(* IEC 61131-3 sources: xPLCCore/codesys_code/Application/COMM_FBs/FB_MpUnpacker, 14 files *)

(* ---- TryReadINTBuffer.st ---- *)
FUNCTION TryReadINTBuffer : POINTER TO BYTE
VAR_INPUT
	sPath 	: STRING; 				  // Path to the integer value
	p_data_size : POINTER TO INT;     // Pointer to an INT to store the size (1, 2, 4, or 8 bytes)
	p_signedness : POINTER TO BOOL;   // Pointer to a BOOL to store if it's signed (TRUE) or unsigned (FALSE)
END_VAR
VAR
	pValue 	: POINTER TO BYTE;    // Pointer to the start of the MessagePack value (type byte)
	tmpByte : BYTE;               // To hold the MessagePack type byte
END_VAR
(* =========== IMPLEMENTATION =========== *)

	// Initialize outputs to default/error states
	IF p_data_size <> 0 THEN
		p_data_size^ := 0; // Default size to 0
	END_IF;
	IF p_signedness <> 0 THEN
		p_signedness^ := FALSE; // Default signedness to FALSE (unsigned)
	END_IF;
	TryReadINTBuffer := 0; // Default return to NULL pointer (no integer found/decoded)

	// Attempt to find the value by path
	IF NOT FindValueByPath(sPath, pValue) THEN
		RETURN; // Value not found, return NULL pointer and default output parameters
	END_IF;

	// Check for NULL pointer from FindValueByPath (should be handled by NOT condition above, but good defense)
	IF pValue = 0 THEN
		RETURN;
	END_IF;

	tmpByte := pValue^; // Read the MessagePack type byte

	// Determine integer type, size, and signedness based on the type byte
	CASE tmpByte OF
		// --- Positive Fixint (0x00 - 0x7F) ---
		0..16#7F: // 0xxxxxxx
			IF p_data_size <> 0 THEN p_data_size^ := 1; END_IF;
			IF p_signedness <> 0 THEN p_signedness^ := TRUE; END_IF; // Can be treated as signed
			TryReadINTBuffer := pValue; // Data is the type byte itself

		// --- Negative Fixint (0xE0 - 0xFF) ---
		16#E0..16#FF: // 111xxxxx
			IF p_data_size <> 0 THEN p_data_size^ := 1; END_IF;
			IF p_signedness <> 0 THEN p_signedness^ := TRUE; END_IF;
			TryReadINTBuffer := pValue; // Data is the type byte itself

		// --- Unsigned Integers ---
		16#CC: // uint 8
			IF p_data_size <> 0 THEN p_data_size^ := 1; END_IF;
			IF p_signedness <> 0 THEN p_signedness^ := FALSE; END_IF;
			TryReadINTBuffer := pValue + 1; // Data starts after the type byte

		16#CD: // uint 16
			IF p_data_size <> 0 THEN p_data_size^ := 2; END_IF;
			IF p_signedness <> 0 THEN p_signedness^ := FALSE; END_IF;
			TryReadINTBuffer := pValue + 1;

		16#CE: // uint 32
			IF p_data_size <> 0 THEN p_data_size^ := 4; END_IF;
			IF p_signedness <> 0 THEN p_signedness^ := FALSE; END_IF;
			TryReadINTBuffer := pValue + 1;

		16#CF: // uint 64
			IF p_data_size <> 0 THEN p_data_size^ := 8; END_IF;
			IF p_signedness <> 0 THEN p_signedness^ := FALSE; END_IF;
			TryReadINTBuffer := pValue + 1;

		// --- Signed Integers ---
		16#D0: // int 8
			IF p_data_size <> 0 THEN p_data_size^ := 1; END_IF;
			IF p_signedness <> 0 THEN p_signedness^ := TRUE; END_IF;
			TryReadINTBuffer := pValue + 1;

		16#D1: // int 16
			IF p_data_size <> 0 THEN p_data_size^ := 2; END_IF;
			IF p_signedness <> 0 THEN p_signedness^ := TRUE; END_IF;
			TryReadINTBuffer := pValue + 1;

		16#D2: // int 32
			IF p_data_size <> 0 THEN p_data_size^ := 4; END_IF;
			IF p_signedness <> 0 THEN p_signedness^ := TRUE; END_IF;
			TryReadINTBuffer := pValue + 1;

		16#D3: // int 64
			IF p_data_size <> 0 THEN p_data_size^ := 8; END_IF;
			IF p_signedness <> 0 THEN p_signedness^ := TRUE; END_IF;
			TryReadINTBuffer := pValue + 1;

		ELSE
			// If not an integer type, return NULL pointer and default output parameters
			// (already set at the beginning of the function)
			TryReadINTBuffer := 0;
	END_CASE;

(* ---- FB_MpUnpacker.st ---- *)
(*
================================================================================
 FB_MpUnpacker: MessagePack Unpacker/Parser with Path Query
================================================================================
This function block parses a MessagePack byte stream.

Instructions:
1. Create a Function Block named 'FB_MpUnpacker'.
2. Copy the main variable declarations into its declaration part.
3. Add each METHOD to the FB, copying the respective variable declarations
   and implementation code.

New Feature: Path Querying
- You can now directly read a value using a path string.
- Use dot notation for nested objects: 'obj.key'
- Use brackets for array indices: 'arr[0]'
- Example: 'data.measurements[2].value'

Key Feature:
- Alignment-Safe: Uses MEMUtils.MemCpy for reading DINT and REAL values
  to prevent memory access violation errors on sensitive hardware.
*)
FUNCTION_BLOCK FB_MpUnpacker
VAR_INPUT
END_VAR
VAR_OUTPUT
	eLastType 		: E_MpType;
	diLastDINT 		: DINT;
	rLastREAL 		: REAL;
	sLastString 	: STRING;
	uiLastCount 	: UINT;
END_VAR
VAR CONSTANT
	MAX_NESTING_DEPTH : INT := 16;
END_VAR
VAR
	pStart 			: POINTER TO BYTE;
	pCurrent 		: POINTER TO BYTE;
	udiSize 		: UDINT;
END_VAR
(* =========== IMPLEMENTATION =========== *)

(* ---- FindValueByPath.st ---- *)
METHOD PRIVATE FindValueByPath : BOOL
VAR_INPUT
	sPath		: STRING;
END_VAR
VAR_IN_OUT
	pResult		: POINTER TO BYTE;
END_VAR
VAR
	sRemainingPath : STRING(255) := sPath;
	sSegment : STRING(80);
	nSepPos, nBracketPos, nEndBracketPos, i, nTargetIndex, nCounter : DINT;
	nMapCount, nArrayCount : UINT;
	sKeyFound : STRING;
	fbTempUnpacker : FB_MpUnpacker;
	// Local pointer for cleaner dereferencing
	pWordLen : POINTER TO WORD; // Declared here
END_VAR
(* =========== IMPLEMENTATION =========== *)
	FindValueByPath := FALSE;
	pResult := pStart;

	WHILE LEN(sRemainingPath) > 0 DO
		IF LEFT(sRemainingPath, 1) <> '[' THEN // This path segment is a key (for a map)
			nSepPos := FIND(sRemainingPath, '.');
			nBracketPos := FIND(sRemainingPath, '[');

			IF nSepPos > 0 AND (nBracketPos = 0 OR nSepPos < nBracketPos) THEN
				sSegment := LEFT(sRemainingPath, DINT_TO_INT(nSepPos - 1));
			ELSIF nBracketPos > 0 AND (nSepPos = 0 OR nBracketPos < nSepPos) THEN
				sSegment := LEFT(sRemainingPath, DINT_TO_INT(nBracketPos - 1));
			ELSE
				sSegment := sRemainingPath;
			END_IF;

			// Handle map header based on marker
			IF (pResult^ >= 16#80 AND pResult^ <= 16#8F) THEN // fixmap
				nMapCount := pResult^ - 16#80;
				pResult := pResult + 1;
			ELSIF pResult^ = 16#DE THEN // map 16
				// --- BUG FIX FOR MAP HEADER ---
				// This was the part still causing issues.
				pWordLen := pResult + 1; // Point to the 2-byte length field
				Swap16To(pWordLen,ADR(nMapCount));
				pResult := pResult + 3; // Advance pointer by 1 (marker) + 2 (count bytes)
			ELSE
				// Current element is not a map, so path segment is invalid
				RETURN;
			END_IF;

			nCounter := 0; // Use nCounter to track if key is found, -1 if found
			FOR i := 1 TO nMapCount DO
				// Initialize a temporary unpacker for the key
				fbTempUnpacker.Init(pResult, udiSize - (pResult - pStart));
				fbTempUnpacker.UnpackNext(); // Unpack the key
				sKeyFound := fbTempUnpacker.sLastString; // Get the key string

				IF NOT SkipValue(pResult) THEN RETURN; END_IF; // pResult now points to the value

				IF sKeyFound = sSegment THEN
					nCounter := -1; // Key found, mark as -1 and exit loop
					EXIT;
				ELSE
					IF NOT SkipValue(pResult) THEN RETURN; END_IF; // Skip the value if key not found
				END_IF;
			END_FOR;

			IF nCounter <> -1 THEN RETURN; END_IF; // If key not found after loop, return FALSE

			sRemainingPath := RIGHT(sRemainingPath, DINT_TO_INT(LEN(sRemainingPath) - LEN(sSegment)));
		ELSE
			nEndBracketPos := FIND(sRemainingPath, ']');
			IF nEndBracketPos = 0 THEN RETURN; END_IF;

			// Extract the index string, e.g., "55" from "[55]"
			sSegment := MID(sRemainingPath, 2, DINT_TO_INT(nEndBracketPos - 2));
			nTargetIndex := STRING_TO_DINT(sSegment);

			// Handle array header based on marker
			IF (pResult^ >= 16#90 AND pResult^ <= 16#9F) THEN // fixarray
				nArrayCount := pResult^ - 16#90;
				pResult := pResult + 1;
			ELSIF pResult^ = 16#DC THEN // array 16
				// --- PREVIOUS BUG FIX FOR ARRAY ---
				pWordLen := pResult + 1; // Point to the 2-byte length field

				Swap16To(pWordLen,ADR(nArrayCount));
				pResult := pResult + 3; // Advance pointer by 1 (marker) + 2 (count bytes)
			ELSE
				// Current element is not an array, so path segment is invalid
				RETURN;
			END_IF;

			// Check if the target index is within the array bounds
			IF nTargetIndex >= DINT_TO_UINT(nArrayCount) THEN RETURN; END_IF;

			// Skip elements until the target index is reached
			FOR i := 0 TO nTargetIndex - 1 DO
				IF NOT SkipValue(pResult) THEN RETURN; END_IF;
			END_FOR;

			sRemainingPath := RIGHT(sRemainingPath, DINT_TO_INT(LEN(sRemainingPath) - nEndBracketPos));

		END_IF;

		IF LEN(sRemainingPath) > 0 AND LEFT(sRemainingPath, 1) = '.' THEN
			sRemainingPath := RIGHT(sRemainingPath, DINT_TO_INT(LEN(sRemainingPath) - 1));
		END_IF;
	END_WHILE;

	FindValueByPath := TRUE;

(* ---- GetValueSize.st ---- *)
METHOD PRIVATE GetValueSize : UDINT
VAR_INPUT
	pObjectStart : POINTER TO BYTE;
END_VAR
VAR
	pTemp : POINTER TO BYTE;
END_VAR
(* =========== IMPLEMENTATION =========== *)
	pTemp := pObjectStart;
	IF SkipValue(pTemp) THEN
		GetValueSize := pTemp - pObjectStart;
	ELSE
		GetValueSize := 0;
	END_IF;

(* ---- Init.st ---- *)
(* Method: Init - (Implementation is unchanged) *)
METHOD Init : BOOL
VAR_INPUT
	pData 		: POINTER TO BYTE;
	udiDataSize : UDINT;
END_VAR
(* =========== IMPLEMENTATION =========== *)
	IF pData = 0 OR udiDataSize = 0 THEN Init := FALSE; RETURN; END_IF;
	pStart 		:= pData;
	pCurrent 	:= pData;
	udiSize 	:= udiDataSize;
	Init 		:= TRUE;

(* ---- SkipValue.st ---- *)
(*
Method: SkipValue [FINAL CORRECTED ITERATIVE VERSION]
Description: Advances a given pointer past the next complete value in the stream.
             This robust iterative version uses a simple counter to avoid recursion
             and correctly handle all MessagePack types.
Return Type: BOOL (TRUE if successful)
*)
METHOD PRIVATE SkipValue : BOOL
VAR_IN_OUT
	pPos : POINTER TO BYTE;
END_VAR
VAR
	diItemsToSkip : DINT := 1; // Start by wanting to skip 1 top-level item.
	byMarker : BYTE;
	udiLength : UDINT;
	uiCount : UINT;
	pWordLen : POINTER TO WORD;

    pDwordLen 	: POINTER TO DWORD;
    udiCount32 	: UDINT;
END_VAR
(* =========== IMPLEMENTATION =========== *)
	WHILE diItemsToSkip > 0 DO
		// Boundary check for each item to be skipped
		IF pPos >= (pStart + udiSize) THEN
			SkipValue := FALSE;
			RETURN;
		END_IF;

		diItemsToSkip := diItemsToSkip - 1; // Consume one item from the "to-skip" list

		byMarker := pPos^; // Read the marker of the current item
		pPos := pPos + 1;  // Advance pointer past the marker

		CASE byMarker OF
    // Nil, Bool, FixInt (0-byte payload, pointer already advanced)
    16#C0, 16#C2, 16#C3: CONTINUE;

    // --- Fixed-size Payloads ---
    16#CC, 16#D0: pPos := pPos + 1; // uint 8, int 8
    16#CD, 16#D1: pPos := pPos + 2; // uint 16, int 16
    16#CE, 16#D2, 16#CA: pPos := pPos + 4; // uint 32, int 32, float 32
    16#CF, 16#D3, 16#CB: pPos := pPos + 8; // uint 64, int 64, float 64

    // --- String Types ---
    16#D9: // str 8
        udiLength := pPos^;
        pPos := pPos + 1 + udiLength;
    16#DA: // str 16
        pWordLen := pPos;
        Swap16To(pWordLen, ADR(udiLength)); // Assumes udiLength gets lower 16 bits
        pPos := pPos + 2 + udiLength;
    16#DB: // str 32
        pDwordLen := pPos;
        Swap32To(pDwordLen, ADR(udiLength)); // Assumes Swap32To helper exists
        pPos := pPos + 4 + udiLength;

    // --- Binary Types ---
    16#C4: // bin 8
        udiLength := pPos^;
        pPos := pPos + 1 + udiLength;
    16#C5: // bin 16
        pWordLen := pPos;
        Swap16To(pWordLen, ADR(udiLength));
        pPos := pPos + 2 + udiLength;
    16#C6: // bin 32
        pDwordLen := pPos;
        Swap32To(pDwordLen, ADR(udiLength));
        pPos := pPos + 4 + udiLength;

    // --- Extension Types ---
    16#D4: pPos := pPos + 2;  // fixext 1 (1-byte type + 1-byte data)
    16#D5: pPos := pPos + 3;  // fixext 2
    16#D6: pPos := pPos + 5;  // fixext 4
    16#D7: pPos := pPos + 9;  // fixext 8
    16#D8: pPos := pPos + 17; // fixext 16
    16#C7: // ext 8
        udiLength := pPos^;
        pPos := pPos + 1 + 1 + udiLength; // len(1) + type(1) + data
    16#C8: // ext 16
        pWordLen := pPos;
        Swap16To(pWordLen, ADR(udiLength));
        pPos := pPos + 2 + 1 + udiLength; // len(2) + type(1) + data
    16#C9: // ext 32
        pDwordLen := pPos;
        Swap32To(pDwordLen, ADR(udiLength));
        pPos := pPos + 4 + 1 + udiLength; // len(4) + type(1) + data

ELSE
    IF (byMarker <= 16#7F) THEN // positive fixint
        CONTINUE;
    ELSIF (byMarker >= 16#E0) THEN // negative fixint
        CONTINUE;

    // fixstr
    ELSIF (byMarker >= 16#A0 AND byMarker <= 16#BF) THEN
        udiLength := byMarker - 16#A0;
        pPos := pPos + udiLength;

    // --- Container Types (add children to skip list) ---
    ELSIF (byMarker >= 16#90 AND byMarker <= 16#9F) THEN // fixarray
        uiCount := byMarker - 16#90;
        diItemsToSkip := diItemsToSkip + uiCount;
    ELSIF (byMarker = 16#DC) THEN // array 16
        pWordLen := pPos;
        Swap16To(pWordLen, ADR(uiCount));
        pPos := pPos + 2;
        diItemsToSkip := diItemsToSkip + uiCount;
    ELSIF (byMarker = 16#DD) THEN // array 32
        pDwordLen := pPos;
        Swap32To(pDwordLen, ADR(udiCount32));
        pPos := pPos + 4;
        diItemsToSkip := diItemsToSkip + udiCount32;

    ELSIF (byMarker >= 16#80 AND byMarker <= 16#8F) THEN // fixmap
        uiCount := (byMarker - 16#80);
        diItemsToSkip := diItemsToSkip + (uiCount * 2);
    ELSIF (byMarker = 16#DE) THEN // map 16
        pWordLen := pPos;
        Swap16To(pWordLen, ADR(uiCount));
        pPos := pPos + 2;
        diItemsToSkip := diItemsToSkip + (uiCount * 2);
    ELSIF (byMarker = 16#DF) THEN // map 32
        pDwordLen := pPos;
        Swap32To(pDwordLen, ADR(udiCount32));
        pPos := pPos + 4;
        diItemsToSkip := diItemsToSkip + (udiCount32 * 2);
    ELSE
        // Unknown marker, cannot safely skip.
        SkipValue := FALSE;
        RETURN;
    END_IF;
END_CASE;

	END_WHILE;

	SkipValue := TRUE;

(* ---- TryReadBool.st ---- *)
METHOD TryReadBool : BOOL
VAR_INPUT
	sPath 	: STRING;
	default : BOOL;
END_VAR
VAR
	pValue : POINTER TO BYTE;
END_VAR
(* =========== IMPLEMENTATION =========== *)
	TryReadBool := default;

	IF FindValueByPath(sPath, pValue) THEN
		IF pValue^ = 16#C2 THEN
			TryReadBool := FALSE;
		ELSIF pValue^ = 16#C3 THEN
			TryReadBool := TRUE;
		END_IF;
	END_IF;

(* ---- TryReadINT64.st ---- *)
METHOD TryReadINT64 : LINT
VAR_INPUT
	sPath 	: STRING; 				// Path to the value
	default 	: LINT; 		// Default value if not found or cannot decode
END_VAR
VAR
	pValue 	: POINTER TO BYTE;
	pCurrent : POINTER TO BYTE; // Pointer to advance through the data
	tmpByte 	: BYTE;
	tmpSint 	: SINT; // For int 8
	tmpWord 	: WORD; // For uint 16, int 16
	tmpInt 	: INT;  // For int 16
	tmpDint 	: DINT; // For uint 32, int 32
	tmpUdint 	: UDINT; // For uint 32
	tmpLint 	: LINT; // For int 64
	tmpULint 	: ULINT; // For uint 64
	// tmpReal : REAL; // Not needed as floats are excluded
	// tmpLReal : LREAL; // Not needed as floats are excluded

	// Define MAX_LINT if not globally available
	cMAX_LINT : LINT := 9223372036854775807; // 2^63 - 1
END_VAR
(* =========== IMPLEMENTATION =========== *)

	TryReadINT64 := default; // Initialize with default value

	IF FindValueByPath(sPath, pValue) THEN
		pCurrent := pValue; // Start at the beginning of the value's data

		// Get the MessagePack type byte
		tmpByte := pCurrent^;
		pCurrent := pCurrent + 1; // Advance pointer past the type byte

		CASE tmpByte OF
			// --- Positive Fixint (0x00 - 0x7F) ---
			0..16#7F: // 0xxxxxxx: Positive Fixint (1 byte)
				TryReadINT64 := BYTE_TO_LINT(tmpByte);

			// --- Negative Fixint (0xE0 - 0xFF) ---
			16#E0..16#FF: // 111xxxxx: Negative Fixint (-32 to -1) (1 byte)
				tmpSint := BYTE_TO_SINT(tmpByte);
				TryReadINT64 := SINT_TO_LINT(tmpSint);

			// --- Unsigned Integers ---
			16#CC: // uint 8 (1 byte value)
				tmpByte := pCurrent^;
				TryReadINT64 := BYTE_TO_LINT(tmpByte);

			16#CD: // uint 16 (2 byte value)
				Swap16To(srcData:=pCurrent, dstData:=ADR(tmpWord));
				TryReadINT64 := WORD_TO_LINT(tmpWord);

			16#CE: // uint 32 (4 byte value)
				Swap32To(srcData:=pCurrent, dstData:=ADR(tmpUdint));
				TryReadINT64 := UDINT_TO_LINT(tmpUdint);

			16#CF: // uint 64 (8 byte value)
				Swap64To(srcData:=pCurrent, dstData:=ADR(tmpULint));
				// Rule: "except (UINT64 && top bit is 1)"
				// This means if tmpULint > MAX_LINT, it cannot be represented as LINT.
				IF tmpULint > cMAX_LINT THEN
					TryReadINT64 := default; // Value too large for signed 64-bit integer
				ELSE
					TryReadINT64 := ULINT_TO_LINT(tmpULint);
				END_IF;

			// --- Signed Integers ---
			16#D0: // int 8 (1 byte value)
				tmpSint := pCurrent^;
				TryReadINT64 := SINT_TO_LINT(tmpSint);

			16#D1: // int 16 (2 byte value)
				Swap16To(srcData:=pCurrent, dstData:=ADR(tmpInt));
				TryReadINT64 := INT_TO_LINT(tmpInt);

			16#D2: // int 32 (4 byte value)
				Swap32To(srcData:=pCurrent, dstData:=ADR(tmpDint));
				TryReadINT64 := DINT_TO_LINT(tmpDint);

			16#D3: // int 64 (8 byte value)
				Swap64To(srcData:=pCurrent, dstData:=ADR(tmpLint));
				TryReadINT64 := tmpLint; // It's already LINT

			// --- Floating-Point Numbers ---
			16#CA, // float 32
			16#CB: // float 64
				// Rule: "they will not read floating point number"
				TryReadINT64 := default; // Explicitly return default for floats

			ELSE
				// Handle other unsupported MessagePack types (string, array, map, nil, ext type)
				TryReadINT64 := default;
		END_CASE;
	END_IF;

(* ---- TryReadObject.st ---- *)
(*
Method: TryReadObject [NEW FEATURE]
Description: Finds a map or array at a given path and initializes a destination
             unpacker instance to represent that sub-object.
Return Type: BOOL (TRUE on success)
*)
METHOD TryReadObject : BOOL
VAR_INPUT
	sPath 	: STRING; 					// Path to the map or array
	pDest 	: POINTER TO FB_MpUnpacker;	// Pointer to the destination unpacker instance
END_VAR
VAR
	pValue : POINTER TO BYTE;
	udiObjectSize : UDINT;
END_VAR
(* =========== IMPLEMENTATION =========== *)
	TryReadObject := FALSE;
	IF pDest = 0 THEN RETURN; END_IF;

	IF FindValueByPath(sPath, pValue) THEN
		IF (pValue^ >= 16#80 AND pValue^ <= 16#8F) OR (pValue^ = 16#DE) OR
		   (pValue^ >= 16#90 AND pValue^ <= 16#9F) OR (pValue^ = 16#DC) THEN
			udiObjectSize := GetValueSize(pObjectStart := pValue);

			IF udiObjectSize > 0 THEN
				TryReadObject := pDest^.Init(pData := pValue, udiDataSize := udiObjectSize);
				TryReadObject:=TRUE;
			END_IF;
		END_IF;
	END_IF;

(* ---- TryReadREAL.st ---- *)
METHOD TryReadREAL : REAL
VAR_INPUT
	sPath 	: STRING; 				// Path to the value
	default 	: REAL; 		// Default value if not found or cannot decode
END_VAR
VAR
	pValue 	: POINTER TO BYTE;
	pCurrent : POINTER TO BYTE; // Pointer to advance through the data
	tmpByte 	: BYTE;
	tmpSint 	: SINT; // For int 8
	tmpWord 	: WORD; // For uint 16, int 16
	tmpInt 	: INT;  // For int 16
	tmpDint 	: DINT; // For uint 32, int 32
	tmpUdint 	: UDINT; // For uint 32
	tmpLint 	: LINT; // For uint 64, int 64
	tmpULint 	: ULINT; // For uint 64
	tmpReal 	: REAL; // For float 32
	tmpLReal 	: LREAL; // For float 64 (double precision)
END_VAR
(* =========== IMPLEMENTATION =========== *)

	TryReadREAL := default; // Initialize with default value

	IF FindValueByPath(sPath, pValue) THEN
		pCurrent := pValue; // Start at the beginning of the value's data

		// Get the MessagePack type byte
		tmpByte := pCurrent^;
		pCurrent := pCurrent + 1; // Advance pointer past the type byte

		// Use a CASE statement for clarity and extensiveness
		CASE tmpByte OF
			// --- Positive Fixint (0x00 - 0x7F) ---
			0..16#7F: // 0xxxxxxx: Positive Fixint (1 byte)
				// The value is directly in tmpByte (pCurrent-1, as pCurrent already advanced)
				TryReadREAL := BYTE_TO_REAL(tmpByte);

			// --- Negative Fixint (0xE0 - 0xFF) ---
			16#E0..16#FF: // 111xxxxx: Negative Fixint (-32 to -1) (1 byte)
				// Treat the byte as SINT (signed 8-bit integer) to get the negative value.
				// tmpByte already holds the value
				tmpSint := BYTE_TO_SINT(tmpByte); // This correctly casts the byte's bits as a signed SINT
				TryReadREAL := SINT_TO_REAL(tmpSint);

			// --- Unsigned Integers ---
			16#CC: // uint 8 (1 byte value)
				tmpByte := pCurrent^; // Read the 1-byte unsigned integer
				TryReadREAL := BYTE_TO_REAL(tmpByte);
				// pCurrent will be implicitly advanced by the next loop iteration or return.

			16#CD: // uint 16 (2 byte value)
				Swap16To(srcData:=pCurrent, dstData:=ADR(tmpWord)); // Swap into tmpWord
				TryReadREAL := WORD_TO_REAL(tmpWord);
				// pCurrent := pCurrent + SIZEOF(WORD); // Already handled implicitly by FindValueByPath or next call

			16#CE: // uint 32 (4 byte value)
				Swap32To(srcData:=pCurrent, dstData:=ADR(tmpUdint)); // Swap into tmpUdint
				TryReadREAL := UDINT_TO_REAL(tmpUdint);
				// pCurrent := pCurrent + SIZEOF(UDINT); // Already handled implicitly

			16#CF: // uint 64 (8 byte value)
				Swap64To(srcData:=pCurrent, dstData:=ADR(tmpULint)); // Swap into tmpULint
				// Conversion from ULINT to REAL might lose precision for very large numbers
				TryReadREAL := ULINT_TO_REAL(tmpULint);
				// pCurrent := pCurrent + SIZEOF(ULINT); // Already handled implicitly

			// --- Signed Integers ---
			16#D0: // int 8 (1 byte value)
				tmpSint := pCurrent^; // Read the 1-byte signed integer
				TryReadREAL := SINT_TO_REAL(tmpSint);
				// pCurrent := pCurrent + SIZEOF(SINT); // Already handled implicitly

			16#D1: // int 16 (2 byte value)
				Swap16To(srcData:=pCurrent, dstData:=ADR(tmpInt)); // Swap into tmpInt
				TryReadREAL := INT_TO_REAL(tmpInt);
				// pCurrent := pCurrent + SIZEOF(INT); // Already handled implicitly

			16#D2: // int 32 (4 byte value)
				Swap32To(srcData:=pCurrent, dstData:=ADR(tmpDint)); // Swap into tmpDint
				TryReadREAL := DINT_TO_REAL(tmpDint);
				// pCurrent := pCurrent + SIZEOF(DINT); // Already handled implicitly

			16#D3: // int 64 (8 byte value)
				Swap64To(srcData:=pCurrent, dstData:=ADR(tmpLint)); // Swap into tmpLint
				// Conversion from LINT to REAL might lose precision for very large numbers
				TryReadREAL := LINT_TO_REAL(tmpLint);
				// pCurrent := pCurrent + SIZEOF(LINT); // Already handled implicitly

			// --- Floating-Point Numbers ---
			16#CA: // float 32 (4 byte value)
				Swap32To(srcData:=pCurrent, dstData:=ADR(tmpReal)); // Swap into tmpReal
				TryReadREAL := tmpReal; // tmpReal now holds the correctly swapped float32
				// pCurrent := pCurrent + SIZEOF(REAL); // Already handled implicitly

			16#CB: // float 64 (8 byte value)
				Swap64To(srcData:=pCurrent, dstData:=ADR(tmpLReal)); // Swap into tmpLReal
				// Convert LREAL to REAL (potential precision loss!)
				TryReadREAL := LREAL_TO_REAL(tmpLReal);
				// pCurrent := pCurrent + SIZEOF(LREAL); // Already handled implicitly

			ELSE
				// Handle unsupported MessagePack types or non-number types gracefully
				// If it's a string, array, map, nil, or ext type, it's not a number and should return the default.
				// Add logging here if needed: 'Unsupported MessagePack type for REAL conversion: %x', tmpByte
				TryReadREAL := default; // Already initialized, but explicitly set for clarity
		END_CASE;
	END_IF;

(* ---- TryReadString.st ---- *)
METHOD TryReadString : STRING
VAR_INPUT
	sPath 		: STRING;
	default 		: STRING;
END_VAR
VAR
	buffer : POINTER TO BYTE;
	buffer_size:UDINT;
END_VAR
(* =========== IMPLEMENTATION =========== *)
	TryReadString := default;

	buffer:=0;
	buffer:=TryReadStringBuffer(sPath,ADR(buffer_size));
	IF(buffer_size>SIZEOF(TryReadString)-1)THEN//and '\0'
		RETURN;
	END_IF
	MEMUtils.MemCpy(ADR(TryReadString),buffer,UDINT_TO_UINT(buffer_size));
	TryReadString[buffer_size]:=0;
	//isOK:=TryReadStringPtr(sPath,ADR(TryReadString),SIZEOF(TryReadString));

(* ---- TryReadStringBuffer.st ---- *)
METHOD TryReadStringBuffer : POINTER TO BYTE
VAR_INPUT
	sPath 		: STRING;
	pStringLength : POINTER TO UDINT; // Pointer to store the extracted string length
END_VAR
VAR
	pItemStart : POINTER TO BYTE;    // Pointer to the start of the MessagePack item (type byte)
	tmpLength  : UDINT;              // Temporary variable for 2-byte or 4-byte string lengths
END_VAR
(* =========== IMPLEMENTATION =========== *)

	TryReadStringBuffer := 0; // Initialize return pointer to NULL

	// Always check if the output pointer is valid before dereferencing
	IF (pStringLength = 0) THEN
		RETURN;
	END_IF;

	// Initialize the output length to 0
	pStringLength^ := 0;

	// Attempt to find the value by path
	IF FindValueByPath(sPath, pItemStart) THEN
		// Check for NULL pointer from FindValueByPath (double-check, though 'IF NOT' covers most cases)
		IF pItemStart = 0 THEN
			RETURN; // Value not found or invalid path
		END_IF;

		// Determine string type based on the first byte (type byte)
		CASE pItemStart^ OF
			// --- Fixstr (0xA0 - 0xBF) ---
			16#A0..16#BF: // 101xxxxx: Fixstr (length is in the lower 5 bits of the type byte)
				pStringLength^ := BYTE_TO_UDINT(pItemStart^ - 16#A0); // Extract length from the type byte
				TryReadStringBuffer := pItemStart + 1; // Content starts after the type byte

			// --- str 8 (0xD9) ---
			16#D9: // 0xD9: str 8 (length is 1 byte)
				pStringLength^ := BYTE_TO_UDINT(pItemStart[1]); // Length is the byte immediately following the type byte
				TryReadStringBuffer := pItemStart + 2; // Content starts after type byte + length byte

			// --- str 16 (0xDA) ---
			16#DA: // 0xDA: str 16 (length is 2 bytes)
				// Swap the 2-byte length from big-endian (MessagePack) to little-endian (CoDeSys)
				Swap16To(srcData:=ADR(pItemStart[1]), dstData:=ADR(tmpLength)); // Swap into temp UDINT
				pStringLength^ := tmpLength; // Assign the (now correctly endian) value
				TryReadStringBuffer := pItemStart + 3; // Content starts after type byte + 2 length bytes

			// --- str 32 (0xDB) ---
			16#DB: // 0xDB: str 32 (length is 4 bytes)
				// Swap the 4-byte length from big-endian (MessagePack) to little-endian (CoDeSys)
				Swap32To(srcData:=ADR(pItemStart[1]), dstData:=ADR(tmpLength)); // Use Swap32To for 4 bytes
				pStringLength^ := tmpLength;
				TryReadStringBuffer := pItemStart + 5; // Content starts after type byte + 4 length bytes

			ELSE
				// If the type byte is not a MessagePack string format,
				// return NULL pointer and 0 length (already initialized at the beginning).
				TryReadStringBuffer := 0;
		END_CASE;
	END_IF;

(* ---- TryReadUINT64.st ---- *)
METHOD TryReadUINT64 : ULINT
VAR_INPUT
	sPath 	: STRING; 				// Path to the value
	default 	: ULINT; 		// Default value if not found or cannot decode
END_VAR
VAR
	pValue 	: POINTER TO BYTE;
	pCurrent : POINTER TO BYTE; // Pointer to advance through the data
	tmpByte 	: BYTE;
	tmpSint 	: SINT; // For int 8
	tmpWord 	: WORD; // For uint 16, int 16
	tmpInt 	: INT;  // For int 16
	tmpDint 	: DINT; // For uint 32, int 32
	tmpUdint 	: UDINT; // For uint 32
	tmpLint 	: LINT; // For int 64
	tmpULint 	: ULINT; // For uint 64
	// tmpReal : REAL; // Not needed as floats are excluded
	// tmpLReal : LREAL; // Not needed as floats are excluded
END_VAR
(* =========== IMPLEMENTATION =========== *)

	TryReadUINT64 := default; // Initialize with default value

	IF FindValueByPath(sPath, pValue) THEN
		pCurrent := pValue; // Start at the beginning of the value's data

		// Get the MessagePack type byte
		tmpByte := pCurrent^;
		pCurrent := pCurrent + 1; // Advance pointer past the type byte

		CASE tmpByte OF
			// --- Positive Fixint (0x00 - 0x7F) ---
			0..16#7F: // 0xxxxxxx: Positive Fixint (1 byte)
				TryReadUINT64 := BYTE_TO_ULINT(tmpByte);

			// --- Negative Fixint (0xE0 - 0xFF) ---
			16#E0..16#FF: // 111xxxxx: Negative Fixint (-32 to -1) (1 byte)
				// Negative numbers cannot be represented as unsigned.
				TryReadUINT64 := default;

			// --- Unsigned Integers ---
			16#CC: // uint 8 (1 byte value)
				tmpByte := pCurrent^;
				TryReadUINT64 := BYTE_TO_ULINT(tmpByte);

			16#CD: // uint 16 (2 byte value)
				Swap16To(srcData:=pCurrent, dstData:=ADR(tmpWord));
				TryReadUINT64 := WORD_TO_ULINT(tmpWord);

			16#CE: // uint 32 (4 byte value)
				Swap32To(srcData:=pCurrent, dstData:=ADR(tmpUdint));
				TryReadUINT64 := UDINT_TO_ULINT(tmpUdint);

			16#CF: // uint 64 (8 byte value)
				Swap64To(srcData:=pCurrent, dstData:=ADR(tmpULint));
				TryReadUINT64 := tmpULint; // It's already ULINT

			// --- Signed Integers ---
			16#D0: // int 8 (1 byte value)
				tmpSint := pCurrent^;
				IF tmpSint < 0 THEN
					TryReadUINT64 := default; // Negative signed int cannot be unsigned
				ELSE
					TryReadUINT64 := SINT_TO_ULINT(tmpSint);
				END_IF;

			16#D1: // int 16 (2 byte value)
				Swap16To(srcData:=pCurrent, dstData:=ADR(tmpInt));
				IF tmpInt < 0 THEN
					TryReadUINT64 := default; // Negative signed int cannot be unsigned
				ELSE
					TryReadUINT64 := INT_TO_ULINT(tmpInt);
				END_IF;

			16#D2: // int 32 (4 byte value)
				Swap32To(srcData:=pCurrent, dstData:=ADR(tmpDint));
				IF tmpDint < 0 THEN
					TryReadUINT64 := default; // Negative signed int cannot be unsigned
				ELSE
					TryReadUINT64 := DINT_TO_ULINT(tmpDint);
				END_IF;

			16#D3: // int 64 (8 byte value)
				Swap64To(srcData:=pCurrent, dstData:=ADR(tmpLint));
				IF tmpLint < 0 THEN
					TryReadUINT64 := default; // Negative signed int cannot be unsigned
				ELSE
					TryReadUINT64 := LINT_TO_ULINT(tmpLint);
				END_IF;

			// --- Floating-Point Numbers ---
			16#CA, // float 32
			16#CB: // float 64
				// Rule: "they will not read floating point number"
				TryReadUINT64 := default; // Explicitly return default for floats

			ELSE
				// Handle other unsupported MessagePack types (string, array, map, nil, ext type)
				TryReadUINT64 := default;
		END_CASE;
	END_IF;

(* ---- UnpackNext.st ---- *)
METHOD UnpackNext : E_MpType
VAR
	byMarker : BYTE;
	udiLength : UDINT;
	diTemp : DINT;
	rTemp : REAL;
	pWordLen : POINTER TO WORD;
	pDwordLen : POINTER TO DWORD;
	// Additional temp variables for big numbers
	tmpByte : BYTE;
	tmpSint : SINT;
	tmpInt : INT;
	tmpWord : WORD;
	tmpUdint : UDINT;
	tmpLint : LINT;
	tmpULint : ULINT;
	tmpLReal : LREAL;
	udiCount32 : UDINT;
END_VAR
(* =========== IMPLEMENTATION =========== *)
eLastType := E_MpType.MP_UNKNOWN;
	UnpackNext := E_MpType.MP_UNKNOWN;

	IF pCurrent >= (pStart + udiSize) THEN RETURN; END_IF;

	byMarker := pCurrent^;
	pCurrent := pCurrent + 1;

	CASE byMarker OF
		// --- Nil ---
		16#C0: eLastType := E_MpType.MP_NIL;

		// --- Boolean ---
		16#C2: eLastType := E_MpType.MP_BOOL; diLastDINT := 0;
		16#C3: eLastType := E_MpType.MP_BOOL; diLastDINT := 1;

		// --- Unsigned Integers ---
		16#CC: // uint 8
			tmpByte := pCurrent^;
			eLastType := E_MpType.MP_DINT; // Store as DINT (fits)
			diLastDINT := BYTE_TO_DINT(tmpByte);
			pCurrent := pCurrent + 1;

		16#CD: // uint 16
			pWordLen := pCurrent;
			Swap16To(pWordLen, ADR(tmpWord));
			eLastType := E_MpType.MP_DINT; // Store as DINT (fits)
			diLastDINT := WORD_TO_DINT(tmpWord);
			pCurrent := pCurrent + 2;

		16#CE: // uint 32
			pDwordLen := pCurrent;
			Swap32To(pDwordLen, ADR(tmpUdint));
			eLastType := E_MpType.MP_DINT; // Store as DINT (may truncate if > 2^31-1)
			IF tmpUdint > 2147483647 THEN // MAX_DINT
				diLastDINT := 2147483647; // Clamp to max DINT
			ELSE
				diLastDINT := UDINT_TO_DINT(tmpUdint);
			END_IF;
			pCurrent := pCurrent + 4;

		16#CF: // uint 64
			Swap64To(srcData:=pCurrent, dstData:=ADR(tmpULint));
			eLastType := E_MpType.MP_DINT; // Store as DINT (will truncate)
			IF tmpULint > 2147483647 THEN // MAX_DINT
				diLastDINT := 2147483647; // Clamp to max DINT
			ELSE
				diLastDINT := ULINT_TO_DINT(tmpULint);
			END_IF;
			pCurrent := pCurrent + 8;

		// --- Signed Integers ---
		16#D0: // int 8
			tmpSint := pCurrent^;
			eLastType := E_MpType.MP_DINT;
			diLastDINT := SINT_TO_DINT(tmpSint);
			pCurrent := pCurrent + 1;

		16#D1: // int 16
			pWordLen := pCurrent;
			Swap16To(pWordLen, ADR(tmpInt));
			eLastType := E_MpType.MP_DINT;
			diLastDINT := INT_TO_DINT(tmpInt);
			pCurrent := pCurrent + 2;

		16#D2: // int 32
			eLastType := E_MpType.MP_DINT;
			MEMUtils.MemCpy(pbyDest:=ADR(diTemp), pbySrc:=pCurrent, dwSize:=SIZEOF(diTemp));
			Swap32To(ADR(diTemp), ADR(diLastDINT));
			pCurrent := pCurrent + 4;

		16#D3: // int 64
			Swap64To(srcData:=pCurrent, dstData:=ADR(tmpLint));
			eLastType := E_MpType.MP_DINT; // Store as DINT (will truncate)
			IF tmpLint > 2147483647 THEN // MAX_DINT
				diLastDINT := 2147483647;
			ELSIF tmpLint < -2147483648 THEN // MIN_DINT
				diLastDINT := -2147483648;
			ELSE
				diLastDINT := LINT_TO_DINT(tmpLint);
			END_IF;
			pCurrent := pCurrent + 8;

		// --- Floating-Point Numbers ---
		16#CA: // float 32
			eLastType := E_MpType.MP_REAL;
			MEMUtils.MemCpy(pbyDest:=ADR(rTemp), pbySrc:=pCurrent, dwSize:=SIZEOF(rTemp));
			Swap32To(ADR(rTemp), ADR(rLastREAL));
			pCurrent := pCurrent + 4;

		16#CB: // float 64
			Swap64To(srcData:=pCurrent, dstData:=ADR(tmpLReal));
			eLastType := E_MpType.MP_REAL; // Convert to REAL (may lose precision)
			rLastREAL := LREAL_TO_REAL(tmpLReal);
			pCurrent := pCurrent + 8;

		// --- String Types ---
		16#D9: // str 8
			udiLength := pCurrent^;
			pCurrent := pCurrent + 1;
			eLastType := E_MpType.MP_STRING;
			MEMUtils.MemCpy(pbyDest:=ADR(sLastString), pbySrc:=pCurrent, dwSize:=UDINT_TO_DWORD(udiLength));
			sLastString[udiLength] := 0;
			pCurrent := pCurrent + udiLength;

		16#DA: // str 16
			pWordLen := pCurrent;
			Swap16To(pWordLen, ADR(udiLength));
			pCurrent := pCurrent + 2;
			eLastType := E_MpType.MP_STRING;
			MEMUtils.MemCpy(pbyDest:=ADR(sLastString), pbySrc:=pCurrent, dwSize:=UDINT_TO_DWORD(udiLength));
			sLastString[udiLength] := 0;
			pCurrent := pCurrent + udiLength;

		16#DB: // str 32
			pDwordLen := pCurrent;
			Swap32To(pDwordLen, ADR(udiLength));
			pCurrent := pCurrent + 4;
			eLastType := E_MpType.MP_STRING;
			// Check if string fits in STRING buffer (typically 255 chars)
			IF udiLength > 255 THEN
				udiLength := 255; // Truncate to max STRING size
			END_IF;
			MEMUtils.MemCpy(pbyDest:=ADR(sLastString), pbySrc:=pCurrent, dwSize:=UDINT_TO_DWORD(udiLength));
			sLastString[udiLength] := 0;
			pCurrent := pCurrent + udiLength;

		// --- Array Types ---
		16#DC: // array 16
			pWordLen := pCurrent;
			Swap16To(pWordLen, ADR(uiLastCount));
			pCurrent := pCurrent + 2;
			eLastType := E_MpType.MP_ARRAY;

		16#DD: // array 32
			pDwordLen := pCurrent;
			Swap32To(pDwordLen, ADR(udiCount32));
			pCurrent := pCurrent + 4;
			eLastType := E_MpType.MP_ARRAY;
			// Store in uiLastCount (may truncate if > 65535)
			IF udiCount32 > 65535 THEN
				uiLastCount := 65535;
			ELSE
				uiLastCount := UDINT_TO_UINT(udiCount32);
			END_IF;

		// --- Map Types ---
		16#DE: // map 16
			pWordLen := pCurrent;
			Swap16To(pWordLen, ADR(uiLastCount));
			pCurrent := pCurrent + 2;
			eLastType := E_MpType.MP_MAP;

		16#DF: // map 32
			pDwordLen := pCurrent;
			Swap32To(pDwordLen, ADR(udiCount32));
			pCurrent := pCurrent + 4;
			eLastType := E_MpType.MP_MAP;
			// Store in uiLastCount (may truncate if > 65535)
			IF udiCount32 > 65535 THEN
				uiLastCount := 65535;
			ELSE
				uiLastCount := UDINT_TO_UINT(udiCount32);
			END_IF;

	ELSE
		// --- Fixint Types (handled in ELSE to catch ranges) ---
		IF (byMarker >= 16#A0 AND byMarker <= 16#BF) THEN // fixstr
			udiLength := byMarker - 16#A0;
			eLastType := E_MpType.MP_STRING;
			MEMUtils.MemCpy(pbyDest:=ADR(sLastString), pbySrc:=pCurrent, dwSize:=UDINT_TO_DWORD(udiLength));
			sLastString[udiLength] := 0;
			pCurrent := pCurrent + udiLength;

		ELSIF (byMarker >= 16#80 AND byMarker <= 16#8F) THEN // fixmap
			eLastType := E_MpType.MP_MAP;
			uiLastCount := byMarker - 16#80;

		ELSIF (byMarker >= 16#90 AND byMarker <= 16#9F) THEN // fixarray
			eLastType := E_MpType.MP_ARRAY;
			uiLastCount := byMarker - 16#90;

		ELSIF (byMarker <= 16#7F) THEN // positive fixint
			eLastType := E_MpType.MP_DINT;
			diLastDINT := BYTE_TO_DINT(byMarker);

		ELSIF (byMarker >= 16#E0) THEN // negative fixint (0xE0-0xFF)
			eLastType := E_MpType.MP_DINT;
			tmpSint := BYTE_TO_SINT(byMarker);
			diLastDINT := SINT_TO_DINT(tmpSint);
		END_IF;
	END_CASE;

	UnpackNext := eLastType;
